FUNCTION_BLOCK FB_04_Start
VAR_INPUT
	bExecute:BOOL;
	bExecute1:BOOL;
END_VAR
VAR_OUTPUT
	bBusy:BOOL;(*功能块执行忙标志*)
	bError:BOOL;(*出错*)
	bDone:BOOL;(*执行完毕*)
END_VAR
VAR_IN_OUT
//	stX:AXIS_REF;
//	stY:AXIS_REF;
//	stZ:AXIS_REF;
	stItpToPlc :NCTOPLC_NCICHANNEL_REF;
	stPlcToItp:PLCTONC_NCICHANNEL_REF;
END_VAR
VAR
	StartStep:INT:=0;
	fbStart:ItpStartStopEx;(*启动和停止*)
END_VAR

CASE StartStep OF
	0:
	  IF  bExecute OR bExecute1 THEN
		 bBusy:=TRUE;(*FB执行状态*)
		 bDone:=FALSE;(*FB执行完毕*)
		 bError:=FALSE;(*报错*)
		 StartStep:=10;(*进入10步*) 
	  END_IF
	10:
	  fbStart(
     	bStart:= bExecute, 
	    bStop:= bExecute1, 
	    tTimeOut:= , 
	    sNciToPlc:= stItpToPlc, 
	    bBusy=> , 
	    bErr=> , 
	    nErrId=> );
	   IF NOT fbStart.bBusy THEN
		  IF NOT fbStart.bErr THEN
			StartStep:=20;(*进入20步*)  
		  ELSE
			bBusy:=FALSE;
			bError:=TRUE;
			StartStep:=999;
		  END_IF
		  fbStart(bStart:= FALSE,bStop:=FALSE,sNciToPlc:= stItpToPlc); 
	    END_IF
	 20:
	   bDone:=TRUE;
       bBusy:=FALSE;   
	   IF NOT bExecute AND NOT bExecute1 THEN
		 StartStep:=0;
	   END_IF
	 999:
	   IF NOT bExecute AND NOT bExecute1 THEN		   
	    StartStep:=0;
        bError:=FALSE; 
	   END_IF
END_CASE

END_FUNCTION_BLOCK

(* stored: Version 1.1.0.1, ProductVersion 3.1.4024.12
   POU FB_04_Start: Id {e563e3e0-6ea4-44dd-90f0-9964064f3104}, SpecialFunc None *)
